Fanuc KAREL source: kf00093.KL

-- PROVISIONAL review KL for V770-1; original PC SHA256 609280debe4402bc17133f105d676a909a79f78a22ccf77e3848dd441457cd18
-- Incomplete behavior may be omitted. Consult companion uncertainty JSON. Do not deploy.
PROGRAM KF00093
%NOLOCKGROUP
VAR
  I : INTEGER
  J : INTEGER
  X : REAL
  Y : REAL
  B : BOOLEAN
  C : BOOLEAN
  TXT : STRING[80]
  TXT2 : STRING[80]
  STATUS : INTEGER
-- UNRESOLVED_DECL AI type=002010
-- UNRESOLVED_DECL BI type=002010
-- UNRESOLVED_DECL P type=000102
-- UNRESOLVED_DECL JP type=000199
-- UNRESOLVED_DECL PF type=000101
-- UNRESOLVED_DECL V1 type=000013
-- UNRESOLVED_DECL V2 type=000013
BEGIN
  -- UNRESOLVED_PC offsets 5-20; opcodes 2E,22,32,35
  -- UNRESOLVED_PC offsets 25-40; opcodes 2E,22,32,35
  -- UNRESOLVED_PC offsets 45-68; opcodes 49,49,94,23
  -- UNRESOLVED_PC offsets 73-77; opcodes 7F
END KF00093
